// TwinCAT 3 PLC project PLC
// ProgramVersion: 3.1.4024.0
// libraries:
//   SPT Base Types, * (Beckhoff Automation LLC)
//   SPT Components, * (Beckhoff Automation LLC)
//   SPT Event Logger, * (Beckhoff Automation LLC)
//   SPT Motion Control, * (Beckhoff Automation LLC)
//   SPT Utilities, * (Beckhoff Automation LLC)
//   Tc2_MC2, * (Beckhoff Automation GmbH)
//   Tc2_MC2_Drive, * (Beckhoff Automation GmbH)
//   Tc2_Standard, * (Beckhoff Automation GmbH)
//   Tc2_System, * (Beckhoff Automation GmbH)
//   Tc3_EventLogger, * (Beckhoff Automation GmbH)
//   Tc3_Module, * (Beckhoff Automation GmbH)
//   Tc3_PackML_V2, * (Beckhoff Automation GmbH)
//   VisuSymbols,3.5.10.0,System
// project tree:
//   DUTs/ MoveState_t.TcDUT
//   / GlobalTextList.TcGTLO, PlcTask.TcTTO, SafetyTask.TcTTO, Visualization Manager.TcVMO (not stored), VISU_TASK.TcTTO
//   GVLs/ GVL_Safety.TcGVL
//   POUs/Components/ FB_GantryXYCylinder.TcPOU, I_Cylinder.TcIO, ST_CylinderX_Command.TcDUT, ST_CylinderX_Config.TcDUT, ST_CylinderX_HMI.TcDUT, ST_CylinderX_Status.TcDUT
//   POUs/ FB_GantryXYZ.TcPOU, FB_Machine.TcPOU, GlobalTextList_1.TcGTLO, MAIN.TcPOU, SAFETY.TcPOU, TestAxis1.TcPOU, TestAxis2.TcPOU
//   VISUs/ V_MachineModule.TcVIS, V_Main.TcVIS, V_Module.TcVIS
// real-time tasks:
//   TASK PlcTask: cycle T#10ms, priority 20, ADS port 350
//   TASK SafetyTask: cycle T#10ms, priority 21, ADS port 351
//   TASK VISU_TASK: cycle T#200000us, priority 30, ADS port 352
// motion (NC):
//   TASK NC-Task 1 SAF: cycle T#2ms, priority 4, ADS port 501
//   TASK NC-Task 1 SVB: cycle T#10ms, priority 8, ADS port 511
//   AXIS Axis 1 (id 1)
//     Dynamic: Acceleration=8053.7925, Deceleration=8053.7925, Jerk=24161.3775
//     Velo: RefSearch=53.69195, RefSync=53.69195, SlowManual=268.45975, FastManual=1610.7585, Fast=5369.195, Maximum=5369.195
//     OtherSettings: AllowMotionCmdToSlave=true
//     encoder EncType=19
//       EncPara: ScaleFactorNumerator=60, ScaleFactorDenominator=1048576, MaxCount=#xffffffff
//     drive DrvType=16
//       DrvPara: MaxCount=#xffffffff, DriveControlDWord=#x00020100
//         Analog: VeloReferenz=5906.1145, VeloScale=32, TorqueSetpointScale=10, ScaleFactorActTorque=0.1
//         TimeComp: TaskDelayCycles=1
//     controller CtrType=1
//       CtrPara: PriorControlFactor=1
//         Observer: BandWidth=20
//   AXIS Axis 2 (id 2)
//     Dynamic: Acceleration=8053.7925, Deceleration=8053.7925, Jerk=24161.3775
//     Velo: RefSearch=53.69195, RefSync=53.69195, SlowManual=268.45975, FastManual=1610.7585, Fast=5369.195, Maximum=5369.195
//     OtherSettings: AllowMotionCmdToSlave=true
//     encoder EncType=19
//       EncPara: ScaleFactorNumerator=60, ScaleFactorDenominator=1048576, MaxCount=#xffffffff
//     drive DrvType=16
//       DrvPara: MaxCount=#xffffffff, DriveControlDWord=#x00020100
//         Analog: VeloReferenz=5906.1145, VeloScale=32, TorqueSetpointScale=10, ScaleFactorActTorque=0.1
//         TimeComp: TaskDelayCycles=1
//     controller CtrType=1
//       CtrPara: PriorControlFactor=1
//         Observer: BandWidth=20
//   AXIS Axis 3 (id 3)
//     Dynamic: Acceleration=8053.7925, Deceleration=8053.7925, Jerk=24161.3775
//     Velo: RefSearch=53.69195, RefSync=53.69195, SlowManual=268.45975, FastManual=1610.7585, Fast=5369.195, Maximum=5369.195
//     OtherSettings: AllowMotionCmdToSlave=true
//     encoder EncType=19
//       EncPara: ScaleFactorNumerator=60, ScaleFactorDenominator=1048576, MaxCount=#xffffffff
//     drive DrvType=16
//       DrvPara: MaxCount=#xffffffff, DriveControlDWord=#x00020100
//         Analog: VeloReferenz=5906.1145, VeloScale=32, TorqueSetpointScale=10, ScaleFactorActTorque=0.1
//         TimeComp: TaskDelayCycles=1
//     controller CtrType=1
//       CtrPara: PriorControlFactor=1
//         Observer: BandWidth=20
// I/O:
//   DEVICE Device 3 (EtherCAT) (disabled), AmsNetId 192.168.1.84.4.1
//     Term 1 (EK1100) [EK1100 EtherCAT Coupler (2A E-Bus)]
//       Term 2 (EL1008) [EL1008 8Ch. Dig. Input 24V, 3ms]
//       Term 3 (EL1008) [EL1008 8Ch. Dig. Input 24V, 3ms]
//       Term 4 (EL2008) [EL2008 8Ch. Dig. Output 24V, 0.5A]
//       Term 5 (EL7221-9014) [EL7221-9014 1Ch. MDP742 Servo motor output stage with OCT (50V, 8A RMS) and STO input]
//         startup 32786:19 := 0000 // DRV Brake Settings / Emergency application timeout
//         startup 32784:51 := 0A00 // DRV Amplifier Settings / Stand still window
//         startup 32785:27 := 01150000 // DRV Motor Settings / Motor speed limitation
//         startup 28688:11 := E803 // DRV Outputs / Torque limitation
//         startup 32784:19 := 5300 // DRV Amplifier Settings / Current loop proportional gain
//         startup 32784:18 := 0500 // DRV Amplifier Settings / Current loop integral time
//         startup 32784:21 := 1F010000 // DRV Amplifier Settings / Velocity loop proportional gain
//         startup 32784:20 := 96000000 // DRV Amplifier Settings / Velocity loop integral time
//         startup 32768:1 := 00 // FB Settings / Invert feedback direction
//       Term 6 (EL7221-9014) [EL7221-9014 1Ch. MDP742 Servo motor output stage with OCT (50V, 8A RMS) and STO input]
//         startup 32785:27 := 01150000 // DRV Motor Settings / Motor speed limitation
//         startup 28688:11 := E803 // DRV Outputs / Torque limitation
//         startup 32784:19 := 5300 // DRV Amplifier Settings / Current loop proportional gain
//         startup 32784:18 := 0500 // DRV Amplifier Settings / Current loop integral time
//         startup 32784:21 := E0000000 // DRV Amplifier Settings / Velocity loop proportional gain
//         startup 32784:20 := 96000000 // DRV Amplifier Settings / Velocity loop integral time
//         startup 32768:1 := 00 // FB Settings / Invert feedback direction
//       Term 7 (EL7221-9014) [EL7221-9014 1Ch. MDP742 Servo motor output stage with OCT (50V, 8A RMS) and STO input]
//         startup 32785:27 := 01150000 // DRV Motor Settings / Motor speed limitation
//         startup 28688:11 := E803 // DRV Outputs / Torque limitation
//         startup 32784:19 := 5300 // DRV Amplifier Settings / Current loop proportional gain
//         startup 32784:18 := 0500 // DRV Amplifier Settings / Current loop integral time
//         startup 32784:21 := E0000000 // DRV Amplifier Settings / Velocity loop proportional gain
//         startup 32784:20 := 96000000 // DRV Amplifier Settings / Velocity loop integral time
//         startup 32768:1 := 00 // FB Settings / Invert feedback direction
//       Term 8 (EL6900) [EL6900, TwinSAFE PLC]
//       Term 9 (EL1904) [EL1904, 4 Ch. Safety Input 24V, TwinSAFE]
//         modules: Module 1 (FSOES)
//       Term 10 (EL2904) [EL2904, 4 Ch. Safety Output 24V, 0.5A, TwinSAFE]
//         modules: Module 1 (FSOES), Module 2 (DO)
//       Term 11 (EL2622) [EL2622 2Ch. Relay Output, NO (230V AC / 30V DC)]
//       Term 12 (EL9011) [EL9011 End Terminal]
// variable links:
//   Device 3 (EtherCAT) <-> Device 3 (EtherCAT)/Term 1 (EK1100)/Term 10 (EL2904)
//     Term 1 (EK1100)/Term 8 (EL6900)/ConnectionInputs/TwinSafeGroup1.Term 10 (EL2904) - Module 1 (FSOES)_3 TxPDO <-> Module 1 (FSOES)/RxPDO/FSOE
//     Term 1 (EK1100)/Term 8 (EL6900)/ConnectionOutputs/TwinSafeGroup1.Term 10 (EL2904) - Module 1 (FSOES)_3 RxPDO <-> Module 1 (FSOES)/TxPDO/FSOE
//   Device 3 (EtherCAT) <-> Device 3 (EtherCAT)/Term 1 (EK1100)/Term 9 (EL1904)
//     Term 1 (EK1100)/Term 8 (EL6900)/ConnectionInputs/TwinSafeGroup1.Term 9 (EL1904) - Module 1 (FSOES)_2 TxPDO <-> Module 1 (FSOES)/RxPDO/FSOE
//     Term 1 (EK1100)/Term 8 (EL6900)/ConnectionOutputs/TwinSafeGroup1.Term 9 (EL1904) - Module 1 (FSOES)_2 RxPDO <-> Module 1 (FSOES)/TxPDO/FSOE
//   NC-Task 1 SAF/Axes/Axis 1 <-> Device 3 (EtherCAT)/Term 1 (EK1100)/Term 5 (EL7221-9014)
//     Drive/Inputs/In/nDataIn1 <-> DRV Following error actual value/Following error actual value
//     Drive/Inputs/In/nDcOutputTime <-> InfoData/DcOutputShift
//     Drive/Inputs/In/nState1 <-> DRV Statusword/Statusword
//     Drive/Inputs/In/nState2 <-> DRV Statusword/Statusword @bit 8
//     Drive/Inputs/In/nState4 @bit 1 <-> WcState/InputToggle
//     Drive/Inputs/In/nState4 <-> WcState/WcState
//     Drive/Outputs/Out/nCtrl1 <-> DRV Controlword/Controlword
//     Drive/Outputs/Out/nCtrl2 <-> DRV Controlword/Controlword @bit 8
//     Drive/Outputs/Out/nDataOut1 <-> DRV Target position/Target position
//     Drive/Outputs/Out/nDataOut2 <-> DRV Target velocity/Target velocity
//     Enc/Inputs/In/nDataIn1 <-> FB Position/Position
//     Enc/Inputs/In/nDcInputTime <-> InfoData/DcInputShift
//     Enc/Inputs/In/nState4 @bit 1 <-> WcState/InputToggle
//     Enc/Inputs/In/nState4 <-> WcState/WcState
//   NC-Task 1 SAF/Axes/Axis 2 <-> Device 3 (EtherCAT)/Term 1 (EK1100)/Term 6 (EL7221-9014)
//     Drive/Inputs/In/nDataIn1 <-> DRV Following error actual value/Following error actual value
//     Drive/Inputs/In/nDataIn3[0] <-> DRV Torque actual value/Torque actual value
//     Drive/Inputs/In/nDcOutputTime <-> InfoData/DcOutputShift
//     Drive/Inputs/In/nState1 <-> DRV Statusword/Statusword
//     Drive/Inputs/In/nState2 <-> DRV Statusword/Statusword @bit 8
//     Drive/Inputs/In/nState4 @bit 1 <-> WcState/InputToggle
//     Drive/Inputs/In/nState4 <-> WcState/WcState
//     Drive/Outputs/Out/nCtrl1 <-> DRV Controlword/Controlword
//     Drive/Outputs/Out/nCtrl2 <-> DRV Controlword/Controlword @bit 8
//     Drive/Outputs/Out/nDataOut1 <-> DRV Target position/Target position
//     Drive/Outputs/Out/nDataOut2 <-> DRV Target velocity/Target velocity
//     Drive/Outputs/Out/nDataOut4 <-> DRV Target torque/Target torque
//     Enc/Inputs/In/nDataIn1 <-> FB Position/Position
//     Enc/Inputs/In/nDataIn3 <-> FB Touch probe 1 pos position/TP1 Pos position
//     Enc/Inputs/In/nDcInputTime <-> InfoData/DcInputShift
//     Enc/Inputs/In/nState4 @bit 1 <-> WcState/InputToggle
//     Enc/Inputs/In/nState4 <-> WcState/WcState
//     Enc/Inputs/In/nState5 <-> FB Touch probe status/Touch probe status/TP1 Enable
//     Enc/Inputs/In/nState6 <-> FB Touch probe status/Touch probe status/TP2 Enable
//     Enc/Inputs/In/nState5 @bit 7 <-> FB Touch probe status/Touch probe status/TP1 Input
//     Enc/Inputs/In/nState6 @bit 7 <-> FB Touch probe status/Touch probe status/TP2 Input
//     Enc/Inputs/In/nState5 @bit 2 <-> FB Touch probe status/Touch probe status/TP1 Neg value stored
//     Enc/Inputs/In/nState6 @bit 2 <-> FB Touch probe status/Touch probe status/TP2 Neg value stored
//     Enc/Inputs/In/nState5 @bit 1 <-> FB Touch probe status/Touch probe status/TP1 Pos value stored
//     Enc/Inputs/In/nState6 @bit 1 <-> FB Touch probe status/Touch probe status/TP2 Pos value stored
//     Enc/Outputs/Out/nCtrl5 @bit 1 <-> FB Touch probe control/Touch probe function/TP1 Continous
//     Enc/Outputs/Out/nCtrl6 @bit 1 <-> FB Touch probe control/Touch probe function/TP2 Continous
//     Enc/Outputs/Out/nCtrl5 <-> FB Touch probe control/Touch probe function/TP1 Enable
//     Enc/Outputs/Out/nCtrl6 <-> FB Touch probe control/Touch probe function/TP2 Enable
//     Enc/Outputs/Out/nCtrl5 @bit 5 <-> FB Touch probe control/Touch probe function/TP1 Enable neg edge
//     Enc/Outputs/Out/nCtrl6 @bit 5 <-> FB Touch probe control/Touch probe function/TP2 Enable neg edge
//     Enc/Outputs/Out/nCtrl5 @bit 4 <-> FB Touch probe control/Touch probe function/TP1 Enable pos edge
//     Enc/Outputs/Out/nCtrl6 @bit 4 <-> FB Touch probe control/Touch probe function/TP2 Enable pos edge
//     Enc/Outputs/Out/nCtrl5 @bit 2 <-> FB Touch probe control/Touch probe function/TP1 Trigger mode
//     Enc/Outputs/Out/nCtrl6 @bit 2 <-> FB Touch probe control/Touch probe function/TP2 Trigger mode
//   NC-Task 1 SAF/Axes/Axis 3 <-> Device 3 (EtherCAT)/Term 1 (EK1100)/Term 7 (EL7221-9014)
//     Drive/Inputs/In/nDataIn1 <-> DRV Following error actual value/Following error actual value
//     Drive/Inputs/In/nDcOutputTime <-> InfoData/DcOutputShift
//     Drive/Inputs/In/nState1 <-> DRV Statusword/Statusword
//     Drive/Inputs/In/nState2 <-> DRV Statusword/Statusword @bit 8
//     Drive/Inputs/In/nState4 @bit 1 <-> WcState/InputToggle
//     Drive/Inputs/In/nState4 <-> WcState/WcState
//     Drive/Outputs/Out/nCtrl1 <-> DRV Controlword/Controlword
//     Drive/Outputs/Out/nCtrl2 <-> DRV Controlword/Controlword @bit 8
//     Drive/Outputs/Out/nDataOut1 <-> DRV Target position/Target position
//     Drive/Outputs/Out/nDataOut2 <-> DRV Target velocity/Target velocity
//     Enc/Inputs/In/nDataIn1 <-> FB Position/Position
//     Enc/Inputs/In/nDcInputTime <-> InfoData/DcInputShift
//     Enc/Inputs/In/nState4 @bit 1 <-> WcState/InputToggle
//     Enc/Inputs/In/nState4 <-> WcState/WcState
//   PLC/PLC Instance <-> Device 3 (EtherCAT)/Term 1 (EK1100)/Term 8 (EL6900)
//     PlcTask Inputs/GVL_Safety.ComError <-> StandardInputs/TwinSafeGroup1.GVL_Safety.ComError_8
//     PlcTask Inputs/GVL_Safety.FBError <-> StandardInputs/TwinSafeGroup1.GVL_Safety.FBError_6
//     PlcTask Inputs/GVL_Safety.SafeError <-> StandardInputs/TwinSafeGroup1.GVL_Safety.SafeError_7
//     PlcTask Outputs/GVL_Safety.ErrorAck <-> StandardOutputs/TwinSafeGroup1.GVL_Safety.ErrorAck_1
//     PlcTask Outputs/GVL_Safety.RunStop <-> StandardOutputs/TwinSafeGroup1.GVL_Safety.RunStop_4
//   PLC/PLC Instance <-> NC-Task 1 SAF/Axes/Axis 1
//     PlcTask Inputs/MAIN.Seedra.GantryXYZ.AxisX.BasicAxis._Axis.NcToPlc <-> Outputs/ToPlc
//     PlcTask Outputs/MAIN.Seedra.GantryXYZ.AxisX.BasicAxis._Axis.PlcToNc <-> Inputs/FromPlc
//   PLC/PLC Instance <-> NC-Task 1 SAF/Axes/Axis 2
//     PlcTask Inputs/MAIN.Seedra.GantryXYZ.AxisY.BasicAxis._Axis.NcToPlc <-> Outputs/ToPlc
//     PlcTask Outputs/MAIN.Seedra.GantryXYZ.AxisY.BasicAxis._Axis.PlcToNc <-> Inputs/FromPlc
//   PLC/PLC Instance <-> NC-Task 1 SAF/Axes/Axis 3
//     PlcTask Inputs/MAIN.Seedra.GantryXYZ.AxisZ.BasicAxis._Axis.NcToPlc <-> Outputs/ToPlc
//     PlcTask Outputs/MAIN.Seedra.GantryXYZ.AxisZ.BasicAxis._Axis.PlcToNc <-> Inputs/FromPlc

CONFIGURATION PLC
    RESOURCE PLC ON TwinCAT3
        TASK PlcTask(INTERVAL := T#10ms, PRIORITY := 20);
        TASK SafetyTask(INTERVAL := T#10ms, PRIORITY := 21);
        TASK VISU_TASK(INTERVAL := T#200000us, PRIORITY := 30);
        PROGRAM MAIN WITH PlcTask : MAIN;
        PROGRAM SAFETY WITH SafetyTask : SAFETY;
        PROGRAM VisuElems_Visu_Prg WITH VISU_TASK : VisuElems.Visu_Prg;
    END_RESOURCE
END_CONFIGURATION

// ---- DUTs/MoveState_t.TcDUT
TYPE MoveState_t :
(
	MOVESTATE_INIT,
	MOVESTATE_ENABLE,
	MOVESTATE_FORWARD,
	MOVESTATE_BACKWARDS,
	MOVESTATE_BACKWARDSSLOW,
	MOVESTATE_NEWTARGETPOSITION,
	MOVESTATE_ERROR,
	MOVESTATE_RESET
);
END_TYPE

// ---- POUs/Components/ST_CylinderX_Command.TcDUT
TYPE ST_CylinderX_Command :
    STRUCT
        RetractExtend  : BOOL;
        RetractCylinder : BOOL;
    END_STRUCT
END_TYPE

// ---- POUs/Components/ST_CylinderX_Config.TcDUT
TYPE ST_CylinderX_Config :
    STRUCT
        ExtendTime  : LREAL;
        RetractTime : LREAL;
    END_STRUCT
END_TYPE

// ---- POUs/Components/ST_CylinderX_HMI.TcDUT
TYPE ST_CylinderX_HMI :
    STRUCT
        Config  : ST_Cylinder_Config;
        Command : ST_CylinderX_Command;
        Status  : ST_CylinderX_Status;
    END_STRUCT
END_TYPE

// ---- POUs/Components/ST_CylinderX_Status.TcDUT
TYPE ST_CylinderX_Status :
    STRUCT
        Extended   : BOOL;
        Retracted  : BOOL;
        Extending  : BOOL;
        Retracting : BOOL;
    END_STRUCT
END_TYPE

// ---- GVLs/GVL_Safety.TcGVL
VAR_GLOBAL
	//State
	SafetySate: INT;
	ErrorAck_RESETED : BOOL;
	
	//TWinSafe Group
	FBError						AT %I* :BOOL; //FBerror
	ComError					AT %I* :BOOL; //ComError
	SafeError					AT %I* :BOOL; //SafeError
	RunStop						AT %Q* :BOOL; //RunStop
	ErrorAck					AT %Q* :BOOL; //ErrorAck
	
	eStopButton					AT %I* :BOOL;
	eStopHMI					:BOOL;
	

	
	//Other
	SAFETY_Permission			AT %I* :BOOL; // FALSE = cannot operate
	RestartFBs_TSG				AT %Q* :BOOL; // Restart FB in TwinSafe Gr //RestartFBs
	
	
END_VAR

// ---- POUs/Components/I_Cylinder.TcIO
INTERFACE I_Cylinder

METHOD Extend
VAR_INPUT
END_VAR
END_METHOD

PROPERTY Extended : BOOL
GET
END_GET
END_PROPERTY

PROPERTY ExtendTime : LREAL
GET
END_GET
SET
END_SET
END_PROPERTY

METHOD Retract
VAR_INPUT
END_VAR
END_METHOD

PROPERTY Retracted : BOOL
GET
END_GET
END_PROPERTY

PROPERTY RetractTime : LREAL
GET
END_GET
SET
END_SET
END_PROPERTY

END_INTERFACE

// ---- POUs/MAIN.TcPOU
PROGRAM MAIN

	VAR
		Seedra          : FB_Machine := (Name := 'SeedraMAIN');
		InitComplete    : BOOL;
	END_VAR

CyclicLogic();

METHOD CyclicLogic
VAR_INPUT
END_VAR
IF NOT InitComplete THEN
    InitComplete := Initialize();
    RETURN;
END_IF

//Machine support HMI & Production Monitor


//Machine Cyclic Logic
Seedra.CyclicLogic();
END_METHOD

METHOD Initialize : BOOL
VAR_INPUT
END_VAR
//Top level machine initialization should happen here, in the main initialization method. Each subsequent "layer" of modules will be named within their respective "parent" intialize method
_AppInfo.KeepOutputsOnBP := TRUE;
Initialize := TRUE;
END_METHOD

END_PROGRAM

// ---- POUs/FB_Machine.TcPOU
FUNCTION_BLOCK FB_Machine EXTENDS FB_PackML_BaseModule // IMPLEMENTS I_ControlsProductionRate
VAR
    // Sub Modules
    GantryXYZ   : FB_GantryXYZ  := (Name := 'Gantry', LogStateChanges := TRUE);

    //Initial List of Components
    ipComponents_Init : ARRAY[1..Parameters_PackML_Base.MAX_NO_OF_COMPONENTS] OF I_ComponentBase := [];

	//Alarms for this module
	MachineAlarms : ARRAY[1..MACHINE_ALARM_COUNT] OF FB_TcAlarm;

END_VAR

VAR CONSTANT
    MACHINE_ALARM_COUNT : INT := 6;
END_VAR


METHOD PROTECTED Clearing
VAR
	i				: UDINT;
	SubModulesReady : BOOL := TRUE;
END_VAR
CASE SequenceState OF
    0:
        NoStateTasksToComplete := FALSE;
        SequenceState          := SequenceState + 10;
    10:
		//Leave Aborted thanks to this
		MachineAlarms[E_Seedra.EmergencyStop].Clear(0, 0);
        SequenceState := SequenceState + 10;
    20:

		SequenceState := SequenceState + 10;
	30: 
	
		SequenceState := SequenceState + 10;
	40:
		StateTasksComplete := TRUE; 
			 
END_CASE

SUPER^.Clearing();
END_METHOD

METHOD PROTECTED CreateEvents
VAR_INPUT
END_VAR
// Add your event creation here
F_CreateAllEventsInClass(Alarms     := MachineAlarms,
                         ClassSize  := SIZEOF(TC_Events.Seedra),
                         pInitEvent := ADR(TC_EVENTS.Seedra.InitReferenceEvent),
                         Prefix     := Name);
// Super call to base
SUPER^.CreateEvents();
END_METHOD

METHOD CyclicLogic
VAR_INPUT
END_VAR

IF NOT _InitComplete THEN
    _InitComplete := Initialize();
    RETURN;
END_IF

SUPER^.CyclicLogic();

//Here the alarms will raise and clear on its own if the input changes

//NOT GVL_Safety.eStopButton -> We Decouple physical button to Activate
  
IF GVL_Safety.eStopHMI OR NOT GVL_Safety.eStopButton AND NOT MachineAlarms[E_Seedra.EmergencyStop].bRaised THEN
	THIS^.ChangeState(E_PMLCommand.ePMLCommand_Abort);
	RaiseAlarmWithStrings(MachineAlarms[E_Seedra.EmergencyStop],'','');
//	ELSIF NOT GVL_Safety.eStop THEN
//	MachineAlarms[E_Seedra.EmergencyStop].Clear(0, 0);

END_IF
END_METHOD

METHOD PROTECTED Execute
CASE _CurrentMode OF

	//=================================PRODUCTION MODE==================================
	E_PMLUnitMode.ePMLUnitMode_Production:
		CASE SequenceState OF
			0:
				NoStateTasksToComplete := FALSE;

				//Advance Gantry to Resetting (Homing)
				GantryXYZ.ChangeState(E_PMLCommand.ePMLCommand_Start);
				
				SequenceState := SequenceState + 10;
					
			10:
				StateTasksComplete := TRUE;
				StateComplete();
				
			
		END_CASE

	//=================================MAINTENANCE & MANUAL MODE==================================
	E_PMLUnitMode.ePMLUnitMode_Maintenance, E_PMLUnitMode.ePMLUnitMode_Manual:
		;
END_CASE
END_METHOD

//! @summary Provides interlocks for HMI control and updates HMI status information for this module
METHOD PROTECTED HMICommunication

//! @description This method is called cyclically by <c>CyclicLogic()</c>

IF GVL_Safety.eStopHMI THEN
	PackMLBaseModule_HMI.Status.Error := TRUE;
	THIS^._Error := TRUE;
END_IF



SUPER^.HMICommunication();
END_METHOD

METHOD PROTECTED HMIPermissions
//General Mode Based Monitoring and handling of HMI control
CASE _CurrentMode OF
   
 E_PMLUnitMode.ePMLUnitMode_Production:
        CASE _CurrentState OF
            E_PMLState.ePMLState_Stopped:
				AllowHMIControl(ThisModuleOnly := FALSE);
            E_PMLState.ePMLState_Idle:
				AllowHMIControl(ThisModuleOnly := FALSE);
            E_PMLState.ePMLState_Suspended:
         		AllowHMIControl(ThisModuleOnly := FALSE);
            E_PMLState.ePMLState_Execute:
            	AllowHMIControl(ThisModuleOnly := FALSE); 
            E_PMLState.ePMLState_Aborted:
                AllowHMIControl(ThisModuleOnly := FALSE); 
            E_PMLState.ePMLState_Held:
                AllowHMIControl(ThisModuleOnly := FALSE); 
            E_PMLState.ePMLState_Complete:
          		AllowHMIControl(ThisModuleOnly := FALSE); 
        END_CASE
		
    E_PMLUnitMode.ePMLUnitMode_Manual:
        AllowHMIControl(ThisModuleOnly := FALSE); 
	E_PMLUnitMode.ePMLUnitMode_Maintenance:
        AllowHMIControl(ThisModuleOnly := FALSE); 
END_CASE
END_METHOD

METHOD PROTECTED Initialize : BOOL
VAR
    i : UDINT; //Generic iteration value
END_VAR
Initialize := FALSE;
CASE DescendantSequenceState OF
    0:
		RegisterSubmodule(GantryXYZ);

        _LogModeChanges         := FALSE;
        _LogStateChanges        := FALSE;
  
	    DescendantSequenceState := DescendantSequenceState + 10;
    10:
        DescendantSequenceState := DescendantSequenceState + 10;
    20:
        //Copy Mode names
        FOR i := 1 TO 3 DO
            ModeNames[i] := F_UnitModeToString(UDINT_TO_DINT(i));
        END_FOR

        DescendantSequenceState := DescendantSequenceState + 10;
    30:
        // Initialize Safety
		IF NOT GVL_Safety.RunStop THEN
			GVL_Safety.RunStop := TRUE;	
		END_IF
        DescendantSequenceState := DescendantSequenceState + 10;
    40:
        //Call the Super
        IF SUPER^.Initialize() THEN
            DescendantSequenceState := DescendantSequenceState + 10;
        END_IF

    50:
        Initialize := TRUE;
END_CASE
END_METHOD

METHOD PROTECTED Resetting
VAR
	i				: UDINT;
	SubModulesReady : BOOL := TRUE;
END_VAR
CASE _CurrentMode OF

	//=================================PRODUCTION MODE==================================
	E_PMLUnitMode.ePMLUnitMode_Production:
		CASE SequenceState OF
			0:
				NoStateTasksToComplete := FALSE;

				//Advance Gantry to Resetting (Homing)
				GantryXYZ.ChangeState(E_PMLCommand.ePMLCommand_Reset);
				
				SequenceState := SequenceState + 10;
					
			10:
				StateTasksComplete := TRUE;
				SUPER^.Resetting();
				
			
		END_CASE

	//=================================MAINTENANCE & MANUAL MODE==================================
	E_PMLUnitMode.ePMLUnitMode_Maintenance, E_PMLUnitMode.ePMLUnitMode_Manual:
		;
END_CASE
END_METHOD

//! @summary This method monitors <b>submodules</b> within this PackML module and initiates fault responses as required
METHOD PROTECTED SubModuleMonitor : BOOL
VAR
	AlarmResponses : ARRAY[0..4] OF E_AlarmResponse; //Temporary response array	
	i			   : UDINT;
END_VAR

//! @description This method is called cyclically by <c>CyclicLogic()</c>
// Check the sub Modules for Alarm Severity
SUPER^.SubModuleMonitor();

//Check the alarms at the machine level
_CurrentAlarmSeverity := F_GetMaxSeverityRaised(Alarms := MachineAlarms, CurrentSeverity := _CurrentAlarmSeverity);

//Check the severity of the machine level alarms
IF _CurrentState <> E_PMLState.ePMLState_Aborted AND _CurrentState <> E_PMLState.ePMLState_Aborting AND _CurrentState <> E_PMLState.ePMLState_Clearing  AND
   _CurrentState <> E_PMLState.ePMLState_Stopped AND _CurrentState <> E_PMLState.ePMLState_Stopping THEN
    AlarmResponses := _ParentFaultResponseDefinitions;
    CASE AlarmResponses[CurrentAlarmSeverity] OF
        E_AlarmResponse.Abort_ImmediateError:
            AbortImmediateError(Name, TRUE);
			AbortImmediateError(Name, FALSE);
        E_AlarmResponse.Abort_Immediate:
            AbortImmediate();
        E_AlarmResponse.Stop_Immediate:
            StopImmediate();
        E_AlarmResponse.Stop_Controlled:
            StopControlled();
        E_AlarmResponse.Hold_Immediate:
            HoldImmediate();
        E_AlarmResponse.Suspend_Immediate:
            SuspendImmediate();
        E_AlarmResponse.Suspend_Controlled:
            SuspendControlled();
        E_AlarmResponse.NoResponse:
            ;
    END_CASE
ELSIF _CurrentState = E_PMLState.ePMLState_Stopped OR _CurrentState = E_PMLState.ePMLState_Stopping THEN
    AlarmResponses := _ParentFaultResponseDefinitions;
    CASE AlarmResponses[CurrentAlarmSeverity] OF
        E_AlarmResponse.Abort_ImmediateError:
            AbortImmediateError(Name, TRUE);
        E_AlarmResponse.Abort_Immediate:
            AbortImmediate();
        E_AlarmResponse.NoResponse:
            ;
    END_CASE
END_IF
END_METHOD

END_FUNCTION_BLOCK

// ---- POUs/FB_GantryXYZ.TcPOU
FUNCTION_BLOCK FB_GantryXYZ EXTENDS FB_PackML_BaseModule 
VAR
    // Sub module definitions here

    // List of sub modules
    ipSubModules_Init : ARRAY[1..Parameters_PackML_Base.MAX_NO_OF_SUBMODULES] OF I_PackML_BaseModule := [];

    // Component definitions here
    AxisX       		: FB_Component_BasicAxis 		:= (Name := 'AxisX');
    AxisY    			: FB_Component_BasicAxis 		:= (Name := 'AxisY');
	AxisZ				: FB_Component_BasicAxis		:= (Name := 'AxisZ');
    GantryCylinder		: FB_GantryXYCylinder			:= (Name := 'Cylinder');
    //Alarms for this module
    GantryAlarms : ARRAY[1..GANTRY_ALARM_COUNT] OF FB_TcAlarm;

	//IO
	LimitSwitchX :BOOL;
	LimitSwitchY :BOOL;
	LimitSwitchZ :BOOL;

	HomeComplete :BOOL;
	
	//resets


END_VAR

VAR CONSTANT
    GANTRY_ALARM_COUNT : INT := 5;
END_VAR


METHOD PROTECTED Aborting
VAR
	i				: UDINT;
	SubModulesReady : BOOL := TRUE;
END_VAR
CASE SequenceState OF
    0:
        NoStateTasksToComplete := FALSE;
        SequenceState          := SequenceState + 10;
    10:
		AxisX.Disable();
		SequenceState := SequenceState + 10;
	20:

		StateTasksComplete := TRUE;
END_CASE

SUPER^.Aborting();
END_METHOD

METHOD PROTECTED Clearing
VAR
	i				: UDINT;
	SubModulesReady : BOOL := TRUE;
END_VAR

VAR_INST
	SoEResetAxis1 : FB_SoEReset;
	ResetAxis1 :	MC_Reset;
END_VAR
CASE SequenceState OF
    0:
        NoStateTasksToComplete := FALSE;
        SequenceState          := SequenceState + 10;
    10:
		//Reset any alarms that get latched
//		GantryAlarms[E_Gantry.AlarmMessage].Clear(0,0);		
//		GantryAlarms[E_Gantry.InfoMessage].Clear(0,0);
//		GantryAlarms[E_Gantry.InitReferenceEvent].Clear(0,0);
//		GantryAlarms[E_Gantry.StartTimeout].Clear(0,0);
//		GantryAlarms[E_Gantry.WarnMessage].Clear(0,0);
//		AxisX.Reset();
//		AxisY.Reset();
//		AxisZ.Reset();



//		AxisX.Reset();

		SoEResetAxis1(Axis := AxisX.Axis);
		SoEResetAxis1.Execute := TRUE;	
		
		ResetAxis1(Axis:=AxisX.Axis);
		ResetAxis1.Execute := TRUE;
		
		
		SequenceState := SequenceState + 10;
	20:
	
		SequenceState := SequenceState + 10;
30: 

		IF NOT ResetSafety() THEN
			ResetSafety();
		ELSE
			SequenceState := SequenceState + 10;	
		END_IF	
    40:

        // Enable here
		// AxisX.Enable();
		// AxisY.Enable();
		// AxisZ.Enable();

        // Check enabled here
		// IF AxisX.Enabled AND AxisY.Enabled AND AxisZ.Enabled THEN
			// SequenceState := SequenceState + 10;
		// END_IF
		
		SequenceState := SequenceState + 10;
		
    50:
        StateTasksComplete := TRUE;
		
END_CASE

SUPER^.Clearing();
END_METHOD

METHOD PROTECTED CreateEvents
VAR_INPUT
END_VAR
// Add your event creation here
F_CreateAllEventsInClass(Alarms     := GantryAlarms,
                         ClassSize  := SIZEOF(TC_EVENTS.Gantry),
                         pInitEvent := ADR(TC_EVENTS.Gantry.InitReferenceEvent),
                         Prefix     := _Name);

// Super call to base
SUPER^.CreateEvents();
END_METHOD

METHOD CuttingBoxFiveSides : BOOL

VAR_INST
	Step : INT ;	
END_VAR



(*
	F			H
	|			|
D---+-----------+---C
	|			|
	|			| 
B---+-----------+---A
	|			|
	E			G
*)
	CASE Step OF
		
		0:  

//Print Info
			
			Trace('Start Cutting Box Five Sides');


			AxisX.MoveVelocity(1,0);
			
			
			Step := Step + 10;	

		10:	//Set Speed

//			AxisX.Velocity := 10; 
//			AxisY.Velocity := 10;
//			AxisZ.Velocity := 5;
			
			Step := Step + 160;

//		20:	//Positioning Motion to A
   			
//			AxisX.MoveAbsolute(0,0);
//			AxisY.MoveAbsolute(250,0);		
			
//			Step := Step + 10; 
		
//		30: //Set Cutting Height
			
//			AxisZ.MoveAbsolute(-30,0);
			
//			Step := Step + 10;

//		40: //Cutting Motion from A to B
			
//			AxisX.MoveAbsolute(500,0);		
			
//			Step := Step + 10;
		
//		50: //Return from Cutting Height 
			
//			AxisZ.MoveAbsolute(50,0);

//			Step := Step + 10;
		
//		60: //Positioning Motion from B to C
			
//			AxisX.MoveAbsolute(0,0);
//			AxisY.MoveAbsolute(50,0);
	
//			Step := Step + 10;

//		70: //Set Cutting Height
		
//			AxisZ.MoveAbsolute(0,0);

//			Step := Step + 10;

//		80: //Cutting Motion from C to D
			
//			AxisX.MoveAbsolute(500,0);
//			AxisY.MoveAbsolute(50,0);

//			Step := Step + 10;

//		90: //Return from Cutting Height 
			
//			AxisZ.MoveAbsolute(50,0);
			
//			Step := Step + 10;

//		100: //Positioning Motion from D to E
			
//			AxisX.MoveAbsolute(450,0);
//			AxisY.MoveAbsolute(300,0);

//			Step := Step + 10;
		
//		110: //Set Cutting Height 	
			
//			AxisZ.MoveAbsolute(0,0);
	
//			Step := Step + 10;

//		120: //Cutting Motion from E to F

//			AxisX.MoveAbsolute(450,0);
//			AxisY.MoveAbsolute(0,0);
			
//			Step := Step + 10;

//		130: //Return from Cutting Height 

//			AxisZ.MoveAbsolute(50,0);
			
//			Step := Step + 10;

//		140: //Positioning Motion from F to G

//			AxisX.MoveAbsolute(50,0);
//			AxisY.MoveAbsolute(300,0);

//			Step := Step + 10;

//		150: //Cutting Motion from G to H
  
//			AxisX.MoveAbsolute(50,0);
//			AxisY.MoveAbsolute(0,0);

//			Step := Step + 10;

//		160: //Return from Cutting Height 
	
//			AxisZ.MoveAbsolute(50,0);

//			Step := Step + 10;

		170: 

//Return to ZERO
////			AxisX.MoveAbsolute(0,0);
//			AxisY.MoveAbsolute(0,0);
			CuttingBoxFiveSides := TRUE;
			Step := 0;
			Trace('Box Five Sides is Cut');
		
			

		

			
	END_CASE
END_METHOD

METHOD CyclicLogic
VAR_INPUT
END_VAR
IF NOT _InitComplete THEN
    _InitComplete := Initialize();
    RETURN;
END_IF

SUPER^.CyclicLogic();

//Set the current alarm severity for this module
_CurrentAlarmSeverity := F_GetMaxSeverityRaised(Alarms := GantryAlarms, CurrentSeverity := _CurrentAlarmSeverity);

//Simulate Alarm Messaging
END_METHOD

METHOD PROTECTED Execute
CASE _CurrentMode OF

	//=================================PRODUCTION MODE==================================
	E_PMLUnitMode.ePMLUnitMode_Production:
		CASE SequenceState OF
			0:
				NoStateTasksToComplete := FALSE;
				
				IF NOT CuttingBoxFiveSides() THEN
					CuttingBoxFiveSides();	
				ELSE
					SequenceState := SequenceState + 10;
				END_IF		
				
			10:		
				StateTasksComplete := TRUE;
				StateComplete();
			END_CASE

	//=================================MAINTENANCE & MANUAL MODE==================================
	E_PMLUnitMode.ePMLUnitMode_Maintenance, E_PMLUnitMode.ePMLUnitMode_Manual:
		;
END_CASE
END_METHOD

METHOD PROTECTED HMIPermissions
//General Mode Based Monitoring and handling of HMI control
CASE _CurrentMode OF
   
 E_PMLUnitMode.ePMLUnitMode_Production:
        CASE _CurrentState OF
            E_PMLState.ePMLState_Stopped:
				AllowHMIControl(ThisModuleOnly := FALSE);
            E_PMLState.ePMLState_Idle:
				AllowHMIControl(ThisModuleOnly := FALSE);
            E_PMLState.ePMLState_Suspended:
         		AllowHMIControl(ThisModuleOnly := FALSE);
            E_PMLState.ePMLState_Execute:
            	AllowHMIControl(ThisModuleOnly := FALSE); 
            E_PMLState.ePMLState_Aborted:
                AllowHMIControl(ThisModuleOnly := FALSE); 
            E_PMLState.ePMLState_Held:
                AllowHMIControl(ThisModuleOnly := FALSE); 
            E_PMLState.ePMLState_Complete:
          		AllowHMIControl(ThisModuleOnly := FALSE); 
        END_CASE
		
    E_PMLUnitMode.ePMLUnitMode_Manual:
        AllowHMIControl(ThisModuleOnly := FALSE); 
	E_PMLUnitMode.ePMLUnitMode_Maintenance:
        AllowHMIControl(ThisModuleOnly := FALSE); 
END_CASE
END_METHOD

METHOD Homing : BOOL

VAR_INST
	Step : INT ;	
END_VAR
CASE Step OF
		
		0: 
			Trace('Enable');
			AxisX.Enable();
		   //AxisX.MoveVelocity(5,0);
			Step := Step + 10; 
		10:
//			Trace('Move Relative');
//			IF IO.DI4 = FALSE THEN
//				AxisX.Home();
//				Step := Step + 10;
//			END_IF
			
//			IF AxisX.Busy = FALSE THEN
//				Step := Step + 10;
//			END_IF
			
			Step := Step + 10;

	
		20:	
			

			Homing := TRUE;
			Step := 0;	

	END_CASE
END_METHOD

//! @summary Basic module initialization logic
METHOD PROTECTED Initialize : BOOL;
VAR
    i                        : UDINT;
    varInfo                  : __SYSTEM.VAR_INFO;
    AllSubUnitsInitialized   : BOOL := TRUE;
    AllComponentsInitialized : BOOL := TRUE;
END_VAR

//! @description This method is called by <c>CyclicLogic()</c> as required
Initialize := FALSE;
CASE DescendantSequenceState OF
    0:
		RegisterComponent(AxisX);
		RegisterComponent(AxisY);	
		RegisterComponent(AxisZ);	
		RegisterComponent(GantryCylinder);
		
        _LogModeChanges         := FALSE;
        _LogStateChanges        := FALSE;
        DescendantSequenceState := DescendantSequenceState + 10;
    10:
        DescendantSequenceState := DescendantSequenceState + 10;
    20:
        //Copy Mode names
        FOR i := 1 TO 3 DO
            ModeNames[i] := F_UnitModeToString(UDINT_TO_DINT(i));
        END_FOR

        DescendantSequenceState := DescendantSequenceState + 10;
    30:
        //Call the Super
        IF SUPER^.Initialize() THEN
            DescendantSequenceState := DescendantSequenceState + 10;
        END_IF
    40:
        Initialize := TRUE;
END_CASE
END_METHOD

METHOD ResetSafety : BOOL
VAR_INST
	Step : INT ;	
	SafetyTimer :TON;
	SafetyTimerTrigger :R_TRIG;
END_VAR
SafetyTimer(IN:= Step > 0 AND NOT SafetyTimer.Q, PT:= T#500MS);

CASE Step OF
		
		0:  // Reset group or waits
			Trace('Timer Initialize');
			Step := Step + 10;
			
		10: //If necessary reset group
		
			GVL_Safety.ErrorAck := (GVL_Safety.ComError OR GVL_Safety.FBError OR GVL_Safety.SafeError); 
		
			IF GVL_Safety.ErrorAck OR SafetyTimer.Q THEN 
				Step := Step + 10;
			END_IF

		20: //Wait for the signal propagation
			IF SafetyTimer.Q THEN
				GVL_Safety.ErrorAck := FALSE;
				Step := Step + 10;
			END_IF
		
		30: //Check FB errors
			IF GVL_Safety.FBError OR (NOT GVL_Safety.SAFETY_Permission) THEN
				GVL_Safety.RestartFBs_TSG := TRUE;
			END_IF
			
			Step := Step + 10;
			
		40: //Wait for the signal propagation
		
			IF SafetyTimer.Q THEN
				GVL_Safety.RestartFBs_TSG := FALSE;
				Step := Step + 10;
			END_IF	
			
		50: //If necessary reset the AX5805
			;
			
		60: //Wait for the signal propagation

			IF SafetyTimer.Q THEN
				
			
			
				IF GVL_Safety.SAFETY_Permission AND 
					NOT (GVL_Safety.ComError OR GVL_Safety.FBError OR GVL_Safety.SafeError) 
				
					THEN
						Step := 0;
						ResetSafety := TRUE;
					ELSE
						Step := 0;
						ResetSafety := FALSE;
				END_IF
			
			END_IF
		
		ELSE
		
		Step := 0;	

END_CASE
END_METHOD

METHOD PROTECTED Resetting
VAR
	i				: UDINT;
	SubModulesReady : BOOL := TRUE;
END_VAR
CASE _CurrentMode OF

	//=================================PRODUCTION MODE==================================
	E_PMLUnitMode.ePMLUnitMode_Production:
		CASE SequenceState OF
			0:
				NoStateTasksToComplete := TRUE;
				
				IF NOT Homing() THEN
					Homing();
				ELSE
					SequenceState := SequenceState + 10;	
				END_IF		
				
			10:		
				StateTasksComplete := TRUE;
				SUPER^.Resetting();
		END_CASE

	//=================================MAINTENANCE & MANUAL MODE==================================
	E_PMLUnitMode.ePMLUnitMode_Maintenance, E_PMLUnitMode.ePMLUnitMode_Manual:
		;
END_CASE
END_METHOD

END_FUNCTION_BLOCK

// ---- POUs/Components/FB_GantryXYCylinder.TcPOU
(*	This FB is used for a single output solenoid 
	It uses the times to say when Extended/Retracted  	
	It starts assuming retracted and the output off.
*)
FUNCTION_BLOCK FB_GantryXYCylinder EXTENDS FB_ComponentBase IMPLEMENTS I_Cylinder
VAR
    //Output
    Output AT %Q* : BOOL;

    // Internal variables
    _ExtendRequest  : BOOL;
    _RetractRequest : BOOL;
    _Extended       : BOOL;
    _Retracted      : BOOL;
    _Extending      : BOOL;
    _Retracting     : BOOL;
    _ExtendTime     : LREAL := 1000; // Default time 1s
    _RetractTime    : LREAL := 1000; // Default time 1s

    // Timer for Extend/Retract
    Extend_TON    : TON;
    Retract_TON   : TON;
    Extend_RTRIG  : R_TRIG;
    Retract_RTRIG : R_TRIG;

    //HMI 
    Cylinder_HMI : ST_CylinderX_HMI;
END_VAR

METHOD PROTECTED CreateEvents
VAR_INPUT
END_VAR
SUPER^.CreateEvents();
END_METHOD

METHOD CyclicLogic
//One shot the requests
Extend_RTRIG(CLK := _ExtendRequest);
Retract_RTRIG(CLK := _RetractRequest);

//Handle Extend
IF Extend_RTRIG.Q THEN
    Output          := TRUE;
    _Extending      := TRUE;
    _Retracting     := FALSE;
    _Retracted      := FALSE;
    _RetractRequest := FALSE;
END_IF

//Handle Retract
IF Retract_RTRIG.Q THEN
    Output         := FALSE;
    _Extending     := FALSE;
    _Retracting    := TRUE;
    _Extended      := FALSE;
    _ExtendRequest := FALSE;
END_IF

//Handle the time to Extend/Retract
Extend_TON(IN := _Extending, PT := LREAL_TO_TIME(_ExtendTime));
Retract_TON(IN := _Retracting, PT := LREAL_TO_TIME(_RetractTime));
IF Extend_TON.Q THEN
    _Extended  := TRUE;
    _Extending := FALSE;
END_IF

IF Retract_TON.Q THEN
    _Retracted  := TRUE;
    _Retracting := FALSE;
END_IF

SUPER^.CyclicLogic();
END_METHOD

METHOD Extend
_ExtendRequest  := TRUE;
_RetractRequest := FALSE;
END_METHOD

PROPERTY Extended : BOOL
GET
Extended := _Extended;
END_GET
END_PROPERTY

PROPERTY ExtendTime : LREAL
GET
ExtendTime := _ExtendTime;
END_GET
SET
END_SET
END_PROPERTY

METHOD PROTECTED HMICommunication
VAR_INPUT
END_VAR
SUPER^.HMICommunication();

//Handle the requests to extend and retract
IF ComponentBase_HMI.Status.HMIControlAvailable THEN
    IF Cylinder_HMI.Command.RetractExtend THEN
        Extend();
    ELSIF Cylinder_HMI.Command.RetractCylinder THEN
        Retract();
    END_IF
END_IF

//Update HMI status info
Cylinder_HMI.Status.Extended    := _Extended;
Cylinder_HMI.Status.Extending   := _Extending;
Cylinder_HMI.Status.Retracted   := _Retracted;
Cylinder_HMI.Status.Retracting  := _Retracting;
Cylinder_HMI.Config.ExtendTime  := _ExtendTime;
Cylinder_HMI.Config.RetractTime := _RetractTime;
END_METHOD

//! @summary Basic component initialization logic
METHOD PROTECTED Initialize : BOOL;

//! @description This method is called by <c>CyclicLogic()</c> as required
//Set the cylinder to retracted
IF Output THEN
    _Extended  := TRUE;
    _Retracted := FALSE;
ELSE
    _Extended  := FALSE;
    _Retracted := TRUE;
END_IF

_Extending      := FALSE;
_ExtendRequest  := FALSE;
_Retracting     := FALSE;
_RetractRequest := FALSE;

//Call base class Initialize
Initialize := SUPER^.Initialize();
END_METHOD

METHOD PROTECTED Monitoring
VAR_INPUT
END_VAR
_Busy    := _Extending OR _Retracting;
_Error   := FALSE;
_ErrorID := 0;
SUPER^.Monitoring();
END_METHOD

METHOD Retract
_ExtendRequest  := FALSE;
_RetractRequest := TRUE;
END_METHOD

PROPERTY Retracted : BOOL
GET
Retracted := _Retracted;
END_GET
END_PROPERTY

PROPERTY RetractTime : LREAL
GET
RetractTime := _RetractTime;
END_GET
SET
_RetractTime := RetractTime;
END_SET
END_PROPERTY

END_FUNCTION_BLOCK

// ---- POUs/SAFETY.TcPOU
PROGRAM SAFETY


//IF GVL_Safety.RUN_STOP = TRUE THEN

//	IF GVL_Safety.SAFETY_Permission = FALSE THEN
	
//		CASE GVL_Safety.SafetySate OF
		
//			0:
//				GVL_Safety.ErrorAck := FALSE;
//				GVL_Safety.SafetySate := GVL_Safety.SafetySate + 10;
//			10:
//				GVL_Safety.ErrorAck := TRUE;
//				GVL_Safety.SafetySate := GVL_Safety.SafetySate + 10;
//			20:
//				GVL_Safety.ErrorAck := FALSE;
//				GVL_Safety.SafetySate := GVL_Safety.SafetySate + 10;
//			30:		
//				GVL_Safety.AX5805_ErrACK := FALSE;
//				GVL_Safety.SafetySate := GVL_Safety.SafetySate + 10;
//			40:	
//				GVL_Safety.AX5805_ErrACK := TRUE;
//				GVL_Safety.SafetySate := GVL_Safety.SafetySate + 10;
//			50:
//				GVL_Safety.AX5805_ErrACK := FALSE;
//				GVL_Safety.SafetySate := GVL_Safety.SafetySate + 10;	
//			60:
//				GVL_Safety.RestartFBs_TSG := FALSE;
//				GVL_Safety.SafetySate := GVL_Safety.SafetySate + 10;
//			70:
//				GVL_Safety.RestartFBs_TSG := TRUE;
//				GVL_Safety.SafetySate := GVL_Safety.SafetySate + 10;	
//			80:
//				GVL_Safety.RestartFBs_TSG := FALSE;
//				GVL_Safety.SafetySate := GVL_Safety.SafetySate + 10;	
//			90:		
//				GVL_Safety.SafetySate := 0;

//		END_CASE
//	END_IF	

//END_IF

END_PROGRAM

// ---- POUs/TestAxis1.TcPOU
FUNCTION_BLOCK TestAxis1
VAR
	
//	Axis1 : AXIS_REF;
//	StateAxis1: MoveState_t;
//	PowerAxis1: MC_Power;
//	Move_Y_MC_Axis1: MC_MoveAbsolute;
//	Move_X_MC_Axis1: MC_MoveAbsolute;
//	ResetAxis1: MC_Reset;
//	HomeAxis1: MC_Home;

//	SoEReadAxis1 : FB_SoERead;
//	SoEResetAxis1 : FB_SoEReset;
	
//	MoveAbsoluteOut1: ST_McOutputs;		(* debug function block output data *)
//	PowerAxis1Out: ST_McOutputs;		(* debug function block output data *)
//	MoveAbsoluteOut2: ST_McOutputs;		(* debug function block output data *)
//	ResetOut : ST_McOutputs;			(* debug function block output data *)

END_VAR

//	(* update the axis status at the beginning of each cycle *)
//		Axis1.ReadStatus();
//		SoEReadAxis1(Axis := Axis1);
//		SoEResetAxis1(Axis := Axis1);
//		PowerAxis1(Axis := Axis1);
//		ResetAxis1(Axis := Axis1);
//		Move_X_MC_Axis1(Axis := Axis1);
//		Move_Y_MC_Axis1(Axis := Axis1);
//		HomeAxis1(Axis := Axis1, bCalibrationCam := IO.DI4);

////IF GVL_Safety.SAFETY_Permission = FALSE THEN

//// resetSafety();

////END_IF		
		
		
//IF GVL_Safety.SAFETY_Permission = TRUE THEN

	
//	(* move axis using a state machine *)
//	CASE StateAxis1 OF

//		MOVESTATE_INIT :	(* initialisation *)
//			(* initialize all function blocks *)
//			Move_X_MC_Axis1.Execute	:= FALSE;
//			Move_Y_MC_Axis1.Execute	:= FALSE;
//			ResetAxis1.Execute		:= FALSE;
//			SoEResetAxis1.Execute 	:= FALSE;
//			StateAxis1				:= MOVESTATE_ENABLE;

//		MOVESTATE_ENABLE :
//			PowerAxis1.Enable := TRUE;
//			PowerAxis1.Enable_Positive := TRUE;
//			PowerAxis1.Enable_Negative := TRUE;
//			HomeAxis1.Execute := TRUE;

//			IF PowerAxis1.Status AND HomeAxis1.Done THEN
//				StateAxis1 := MOVESTATE_FORWARD;
//			ELSIF PowerAxis1.Error THEN
//				StateAxis1 := MOVESTATE_ERROR;
//			END_IF

//		MOVESTATE_FORWARD :		(* start to first position *)
//			Move_X_MC_Axis1.Position := 1500;		(* start to intermediate tartet position *)
//			Move_X_MC_Axis1.Velocity := 1500;		(* medium velocity level *)
//			Move_X_MC_Axis1.BufferMode := MC_Buffered;
//			Move_X_MC_Axis1.Execute := TRUE;
//			IF Move_X_MC_Axis1.Active  THEN
//				(* axis is executing job but is not yet finished *)
//				Move_X_MC_Axis1.Execute := FALSE;
//				(* leave this state and buffer a second command *)
//				StateAxis1 := MOVESTATE_NEWTARGETPOSITION;
//			ELSIF Move_X_MC_Axis1.CommandAborted OR Move_X_MC_Axis1.Error THEN
//				StateAxis1 := MOVESTATE_ERROR;
//			END_IF

//		MOVESTATE_NEWTARGETPOSITION :		(* change target position while moving *)
//			(* start a buffered motion command while axis is moving *)
//			Move_Y_MC_Axis1.Position := 5000;		(* start to final target *)
//			Move_Y_MC_Axis1.Velocity := 2000;		(* increase velocity *)
//			Move_Y_MC_Axis1.BufferMode := MC_BlendingPrevious; 	(* use velocity of previous command till intermediate target position position *)
//			Move_Y_MC_Axis1.Execute := TRUE;
//			IF Move_Y_MC_Axis1.Done THEN
//				Move_Y_MC_Axis1.Execute := FALSE;
//				StateAxis1 := MOVESTATE_BACKWARDS;
//			ELSIF Move_Y_MC_Axis1.CommandAborted OR Move_Y_MC_Axis1.Error THEN
//				StateAxis1 := MOVESTATE_ERROR;
//			END_IF

//		MOVESTATE_BACKWARDS :	(* move back to initial position *)
//			Move_X_MC_Axis1.Position := 100;		(* position close to initial position *)
//			Move_X_MC_Axis1.Velocity := 50;		(* high velocity *)
//			Move_X_MC_Axis1.BufferMode := MC_Buffered;
//			Move_X_MC_Axis1.Execute := TRUE;
//			IF Move_X_MC_Axis1.Active THEN
//				(* axis is executing job but is not yet finished *)
//				Move_X_MC_Axis1.Execute := FALSE;
//				(* leave this state and buffer a second command *)
//				StateAxis1 := MOVESTATE_BACKWARDSSLOW;
//			ELSIF Move_X_MC_Axis1.CommandAborted OR Move_X_MC_Axis1.Error THEN
//				StateAxis1 := MOVESTATE_ERROR;
//			END_IF

//		MOVESTATE_BACKWARDSSLOW :	(* move back to initial position *)
//			(* start a buffered motion command while axis is moving *)
//			Move_Y_MC_Axis1.Position := 0;	(* back to initial position *)
//			Move_Y_MC_Axis1.Velocity := 50; 	(* slow velocity *)
//			Move_Y_MC_Axis1.BufferMode := MC_BlendingNext; 	(* use velocity from first target position *)
//			Move_Y_MC_Axis1.Execute := TRUE;
//			IF Move_Y_MC_Axis1.Done THEN
//				Move_Y_MC_Axis1.Execute := FALSE;
//				StateAxis1 := MOVESTATE_FORWARD;
//			ELSIF Move_Y_MC_Axis1.CommandAborted OR Move_Y_MC_Axis1.Error THEN
//				StateAxis1 := MOVESTATE_ERROR;
//			END_IF

//		MOVESTATE_ERROR :
//			IF Axis1.Status.Error OR SoEReadAxis1.Error THEN
//				StateAxis1 := MOVESTATE_RESET;	(* axis error re quires reset *)
//			ELSE 
//				StateAxis1 := MOVESTATE_INIT;		(* function block errors don't need a reset *)
//			END_IF

//		MOVESTATE_RESET :
//			ResetAxis1.Execute := TRUE; 		
//			SoEResetAxis1.Execute := TRUE;
//			IF ResetAxis1.Done THEN
//				StateAxis1 := MOVESTATE_INIT;
//			ELSIF ResetAxis1.Error THEN
//				StateAxis1 := MOVESTATE_INIT; (* can't do anything here *)
//			END_IF

//	END_CASE

//END_IF

END_FUNCTION_BLOCK

// ---- POUs/TestAxis2.TcPOU
FUNCTION_BLOCK TestAxis2 EXTENDS FB_ComponentBase
VAR
	AxisSPT : FB_BasicAxis;
	State 	: INT;
END_VAR

METHOD PUBLIC CyclicLogic
VAR	

END_VAR
SUPER^.CyclicLogic();
END_METHOD

METHOD PROTECTED Initialize : BOOL;
SUPER^.Initialize();
END_METHOD

METHOD MoveAxis
      AxisSPT.CyclicLogic();

IF GVL_Safety.SAFETY_Permission = TRUE THEN

	CASE State OF
		
	00:
		IF AxisSPT.Enable() THEN
			State := State + 10;
		END_IF
	10:
		IF AxisSPT.Enabled THEN
			AxisSPT.MoveVelocity( -5, TRUE);	
		
			IF IOx.DI4 = TRUE THEN
				AxisSPT.Home();
				State := State + 10;
			END_IF
		END_IF

	
	20:
		AxisSPT.Velocity := 10;
		IF AxisSPT.MoveAbsolute(5000, FALSE) THEN
			State := State + 10;
		END_IF

	30:
		IF NOT AxisSPT.Busy THEN
			State := State + 10;
		END_IF

	40:
		AxisSPT.Trace('****Done****'); 

	50:
		//

	END_CASE

END_IF
END_METHOD

END_FUNCTION_BLOCK

// ---- GlobalTextList.TcGTLO
TEXTLIST GlobalTextList
  452 = 'Clear'
  46 = 'Maintenance'
  904 = 'Manual'
  929 = 'Production'
  181 = 'Reset'
  77 = 'Start'
  516 = 'State: %s'
  98 = 'STOP'
END_TEXTLIST

// ---- POUs/GlobalTextList_1.TcGTLO
TEXTLIST GlobalTextList_1
  685 = '%s'
  470 = '>'
  680 = 'Abort'
  10 = 'ANIHILATIOn'
  621 = 'ANIHILATION'
  347 = 'BB8'
  452 = 'Clear'
  424 = 'EStop'
  744 = 'Hold'
  46 = 'Maintenance'
  904 = 'Manual'
  929 = 'Production'
  181 = 'Reset'
  77 = 'Start'
  354 = 'START'
  516 = 'State: %s'
  828 = 'Stop'
  98 = 'STOP'
  806 = 'Suspend'
  197 = 'Unhold'
  832 = 'Unsuspend'
  500 = 'V'
  277 = '▶'
  821 = '▶\nStart'
  266 = '▶Start'
END_TEXTLIST

// ---- VISUs/V_MachineModule.TcVIS
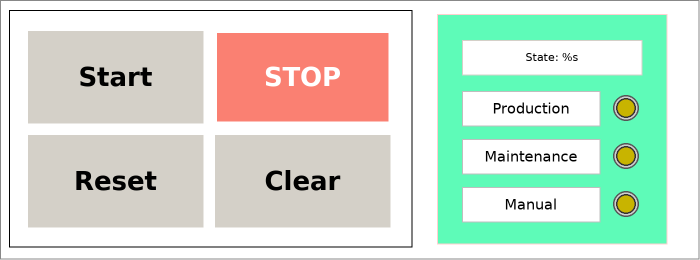
VISUALIZATION V_MachineModule  // 700x260
VAR_IN_OUT
	HMI : ST_PackMLBaseModule_HMI;
END_VAR
    Frame (432,10 240x240)
        shows V_Module(HMI := HMI)
    RoundedRectangle (9,10 403x237)
    RoundedRectangle (28,31 175x92), "Start"
        OnMouseClick: execute { HMI.Command.State := E_PMLCommand.ePMLCommand_Start; }
    RoundedRectangle (215,135 175x92), "Clear"
        OnMouseClick: execute { HMI.Command.State := E_PMLCommand.ePMLCommand_Clear; }
    RoundedRectangle (28,135 175x92), "Reset"
        OnMouseClick: execute { HMI.Command.State := E_PMLCommand.ePMLCommand_Reset; }
    RoundedRectangle (215,31 175x92), "STOP"
        toggle GVL_Safety.eStopHMI
        OnMouseClick: execute {  }
END_VISUALIZATION

// ---- VISUs/V_Main.TcVIS
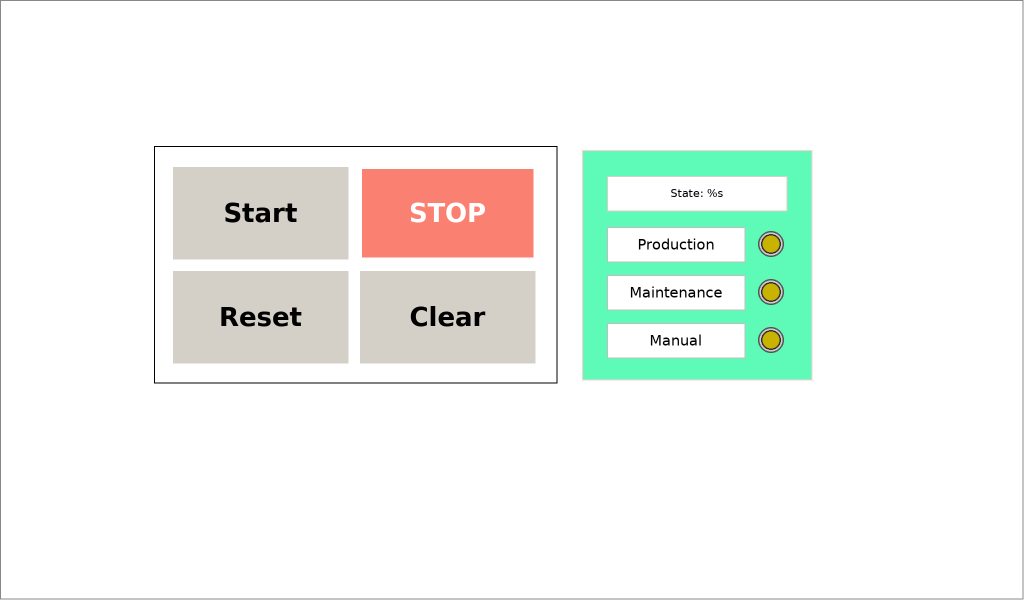
VISUALIZATION V_Main  // 1024x600
    Frame (145,136 700x260)
        shows V_MachineModule(HMI := MAIN.Seedra.PackMLBaseModule_HMI)
END_VISUALIZATION

// ---- VISUs/V_Module.TcVIS
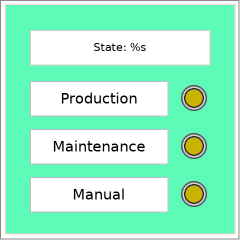
VISUALIZATION V_Module  // 240x240
VAR_IN_OUT
	HMI : ST_PackMLBaseModule_HMI;
END_VAR
    RoundedRectangle (5,4 230x230)
    Textfield (30,30 180x35), "State: %s", text variable: HMI.Status.State
    Lamp1 (179,83 30x30), variable: HMI.Status.Mode = E_PMLUnitMode.ePMLUnitMode_Production, style: Lamp-Lamp1-Yellow
    Lamp1 (179,131 30x30), variable: HMI.Status.Mode = E_PMLUnitMode.ePMLUnitMode_Maintenance, style: Lamp-Lamp1-Yellow
    Lamp1 (179,179 30x30), variable: HMI.Status.Mode = E_PMLUnitMode.ePMLUnitMode_Manual, style: Lamp-Lamp1-Yellow
    RoundedRectangle (30,81 138x35), "Production"
        OnMouseClick: execute { HMI.Command.Mode := E_PMLUnitMode.ePMLUnitMode_Production; }
    RoundedRectangle (30,129 138x35), "Maintenance"
        OnMouseClick: execute { HMI.Command.Mode := E_PMLUnitMode.ePMLUnitMode_Maintenance; }
    RoundedRectangle (30,177 138x35), "Manual"
        OnMouseClick: execute { HMI.Command.Mode := E_PMLUnitMode.ePMLUnitMode_Manual; }
END_VISUALIZATION
